# EPICS substitutions: dg645App/Db/dg645Ch.substitutions
file dg645Ch.template {
pattern
{CHAN, REF}
{   0,   0}
{   1,   0}
{   2,   0}
{   3,   2}
{   4,   0}
{   5,   4}
{   6,   0}
{   7,   6}
{   8,   0}
{   9,   8}
}
